(* IEC 61131-3 sources: ArfBotOS/Codesys-4/ArfBotOS.fbsdev/Application.iecapp^/FUN/home/FB_HomingProcessor.fb.st^/private, 1 file *)

(* ---- _M_HandlePose.meth.st ---- *)
METHOD PRIVATE _M_HandlePose : BOOL
VAR_IN_OUT
	AxisGroup: AXIS_GROUP_REF_SM3;
	GroupHandler: FB_GroupHandler;
END_VAR
VAR_INPUT
END_VAR
VAR
	_MoveCommand: ST_MoveCmd;
	_PoseSpeed: LREAL:=20.0;
END_VAR

IF _MoveToPose THEN
	_MoveToPose:= FALSE;
	//
	IF GVL_App.Enable
		AND_THEN Flags[GVL_App.HOME_COMPLETE].Value
		AND_THEN NOT _MoveCommandProcessor.Busy
		AND_THEN NOT _MoveCommandProcessor.Error THEN
			//
			_MoveCommand.MoveType 			:= DUT_Command_MoveType.DirectMove;
			_MoveCommand.PositionType 		:= DUT_Command_PositionType.AbsolutePosition;
			_MoveCommand.CoordinateType 	:= DUT_Command_CoordinateType.Literal;
			_MoveCommand.Speed 				:= _PoseSpeed;
			_MoveCommand.CoordSystem 		:= SMC_COORD_SYSTEM.ACS;
			_MoveCommand.CoordRef 			:= StoredPositions[GVL_App.POSE_2_IDX].Position;
			//
			_MoveCommandProcessor.Command := F_BuildMoveCmd(_MoveCommand);
			_MoveCommandProcessor.M_Start();
	END_IF;
END_IF

_MoveCommandProcessor(
	StoredPositions:= StoredPositions,
	VisionRegisters:= VisionRegisters,
	Flags:= Flags,
	AxisGroup:= AxisGroup,
	GroupHandler:= GroupHandler,
	Velocity:= StoredPositions[GVL_App.SPEEDS_IDX].Position.X,
	VelFactor:= StoredPositions[GVL_App.SPEEDS_IDX].Position.A,
	Acceleration:= StoredPositions[GVL_App.SPEEDS_IDX].Position.Y,
	AccFactor:= StoredPositions[GVL_App.SPEEDS_IDX].Position.B,
	Jerk:= StoredPositions[GVL_App.SPEEDS_IDX].Position.Z,
	JerkFactor:= StoredPositions[GVL_App.SPEEDS_IDX].Position.C,
	Position=> ,
	ItfUnitMode=> ,
	Error=> );
END_METHOD
